// TIA Portal V19 export
VAR_GLOBAL   // PLC tag table "Default tag table"
   Tag_1 AT %M3.0 : Bool;
   Tag_2 AT %M1.0 : Bool;
END_VAR
